# EPICS substitutions: ngpspsuSup/current_and_voltage.substitutions
file current_and_voltage.template {

pattern {P, PORT, RNAME, TITLE_NAME, LOWER_NAME, UNITS}
{"\$(P)", \$(PORT), "VOLT", "Voltage", "voltage", "V" }
{"\$(P)", \$(PORT), "CURR", "Current", "current", "A" }
}
